FUNCTION_BLOCK FB_TempSensPtx IMPLEMENTS I_TemperatureSensor
(*Classic Pt temperature sensor. The ConvFac defines the resulting Pt sensor (i.e. ConvFac=100 -> Pt100).
Measurement is directly converted into °C.*)
VAR_OUTPUT
END_VAR
VAR
	ConvFac : INT := 10; // Conversion factor (for Pt100 this is 100, Pt1000 it`s 1000, ..)
	fTemperature : REAL; // Properties
	TempRaw AT %I* : INT; // Raw value
END_VAR

METHOD FB_init : BOOL
VAR_INPUT
	bInitRetains : BOOL; // if TRUE, the retain variables are initialized (warm start / cold start)
	bInCopyCode : BOOL;  // if TRUE, the instance afterwards gets moved into the copy code (online change)
	Ptx : INT := 100; // x value (for Pt100 this is 100, Pt1000 it`s 1000, ..)
END_VAR
ConvFac := Ptx/10; // Divide by ten to get conversion factor
END_METHOD

METHOD Run
fTemperature := INT_TO_REAL(TempRaw)/ConvFac; // Read and convert raw temperature measurement
END_METHOD

PROPERTY Temperature : REAL
GET
Temperature := THIS^.fTemperature;
END_GET
SET
END_SET
END_PROPERTY

END_FUNCTION_BLOCK

(* stored: Version 1.1.0.1, ProductVersion 3.1.4024.6
   POU FB_TempSensPtx: Id {1001b5c2-46d4-4dfc-9afb-b99f84f108f9}, SpecialFunc None
   Method FB_init: Id {31b8d0d5-2b72-4ea3-a7e5-c44bc48a1e69}
   Method Run: Id {f7d5f006-fab3-4a4c-a463-dd18f2f325e1}
   Property Temperature: Id {cc870965-0066-4233-95bf-a193f6d65dc5}
   Get Get: Id {a7dddca7-b9b6-4793-8a13-6705664706bc}
   Set Set: Id {247fbcc2-7a1a-4b6f-94ee-05fbd6afef1f} *)
